FUNCTION_BLOCK FB_AnnealingOvenSealingSystem EXTENDS FB_SystemContinous
VAR_INPUT
END_VAR
VAR_OUTPUT
END_VAR
VAR
	//default parameters
	localDefaultParameters : ST_AnnealingOvenExhaustGasDefaultParameters;

	//pumps
	stPU261DefaultParameters : ST_PumpGrundfosMagna3DefaultParameters := (bPumpBeforeApplication := FALSE, tTaskCycleTime := GlobalVariables.tTaskCycleTime_MAIN, tCtrlCycleTime := GlobalVariables.tCtrlCycleTime_MAIN);
	PU261 : FB_PumpGrundfosMagna3 := (ST_DefaultParameters := stPU261DefaultParameters);

	//valves
	stRV261DefaultParameters : ST_MixingValveDefaultParameters := (bFeedbackSignal := TRUE, tTaskCycleTime := GlobalVariables.tCtrlCycleTime_MAIN, tCtrlCycleTime := GlobalVariables.tCtrlCycleTime_MAIN);
	RV261 : FB_MixingValve := (ST_DefaultParameters := stRV261DefaultParameters);
	
	//sensors	
	WMZ261 : FB_MollineC3HeatCounter;
	
	//internal variables
	bSetStatusOn_PU261 : BOOL;
	bSetStatusOn_RV261 : BOOL;
END_VAR

MAIN();

//pumps
PU261.GetState_Profibus();
PU261(bSetStatusOnAutomatic := bSetStatusOn_PU261,
	fSetPointAutomatic := fSetPoint,
	bAlgorithmPermission := bAlgorithmPermission,
	nControlModeAutomatic := 2);
PU261.SetState_Profibus();

//valves
RV261.GetState_AI();
RV261(bSetStatusOnAutomatic := bSetStatusOn_RV261,
	fSetPointAutomatic := 100,
	bAlgorithmPermission := bAlgorithmPermission,
	nControlModeAutomatic := 0);
RV261.SetState_AO();

WMZ261(aHeatCounterTelegramm := Telegramm_WZ_Ofenkuehlung);

METHOD PROTECTED  CheckError : BOOL
VAR_INPUT
END_VAR
VAR_OUTPUT
	bError : BOOL;
END_VAR
bError := PU261.bError;
END_METHOD

METHOD PROTECTED  Operational : BOOL
VAR_INPUT
END_VAR
VAR_OUTPUT
	bSwitchToWorking : BOOL := FALSE;
END_VAR
bSetStatusOn_PU261 := TRUE;

IF PU261.bStatusOn THEN
	bSwitchToWorking := TRUE;
END_IF
END_METHOD

METHOD PROTECTED  RampDown : BOOL
VAR_INPUT
END_VAR
VAR_OUTPUT
	bRampDownFinished : BOOL := FALSE;
END_VAR
bSetStatusOn_PU261 := FALSE;

IF NOT PU261.bStatusOn THEN
	bSetStatusOn_RV261 := FALSE;
	IF RV261.fOperatingPoint<10 THEN
		bRampDownFinished := TRUE;
	END_IF
END_IF
END_METHOD

METHOD PROTECTED  RampUp : BOOL
VAR_INPUT
END_VAR
VAR_OUTPUT
	bRampUpFinished : BOOL := FALSE;
END_VAR
bSetStatusOn_RV261 := TRUE;
bRampUpFinished := TRUE;
END_METHOD

METHOD PROTECTED   SetSetPointLimits : BOOL
VAR_INPUT
END_VAR
aSetPointLimits[1] := localDefaultParameters.aSetPointLimitsTemperature[1];
aSetPointLimits[2] := localDefaultParameters.aSetPointLimitsTemperature[2];
END_METHOD

METHOD PROTECTED  SetState : BOOL
VAR_INPUT
END_VAR
VAR_OUTPUT
END_VAR
fOperatingPoint := PU261.fTemperatureInternal;

controlState.bStatusOn := bSetStatusOn;
setPointState.aSetPointLimits := aSetPointLimits;
setPointState.fSetPoint := fSetPoint;
setPointState.fOperatingPoint := fOperatingPoint;
setPointState.sSetPointUnit := 'degreeC';
setPointState.sOperatingPointUnit := 'degreeC';
END_METHOD

METHOD PROTECTED  Working : BOOL
VAR_INPUT
END_VAR
VAR_OUTPUT
	bSwitchToOperational : BOOL := FALSE;
END_VAR
//empty method
END_METHOD

END_FUNCTION_BLOCK

(* stored: Version 1.1.0.1, ProductVersion 3.1.4024.10
   POU FB_AnnealingOvenSealingSystem: Id {c79fb180-c52a-479d-9180-03a928329c11}, SpecialFunc None
   Method CheckError: Id {0884511a-7c08-4815-9766-3acf5bdad9b7}
   Method Operational: Id {3b8fc09c-a3eb-4e29-a806-30ced16dbd57}
   Method RampDown: Id {19a3e988-adfd-4643-8b51-813eea489db5}
   Method RampUp: Id {7093dcc9-6881-4082-97ed-41554badcf83}
   Method SetSetPointLimits: Id {06ca703d-33d0-4427-9c5b-35d2baa1d962}
   Method SetState: Id {094fc672-9f27-4d6a-bd6e-224fcaf867d0}
   Method Working: Id {50b4e403-2e2a-4fdc-86ac-77113ce6f10b} *)
